CASE outputState OF
	eSpecialStates.SLAVE_ENTER_PROCEDURE:
		bSerialTransition := clamper^.Execute(eCylinderCommands.COMMAND_B); //release
	16#201:
		//wait until trigger off
		bSerialTransition := NOT handy;
		IF bSerialTransition THEN
			SlotBase^.Valid := FALSE; //reset
		END_IF
		//
		IF toggleClear AND materialRemains = 0 THEN
			toggleClear := FALSE;
		END_IF
	16#202:
		//conditions
		//1. bypassed
		//2. handy on
		//3. toggle clear
		//4. material existed with light screen off
		IF toggleClear OR bIsBypassed OR handy OR ( lightScreen AND SlotBase^.Valid) THEN
			bSerialTransition := TRUE;
		END_IF
		//once material detected , clamper imdiatly
		IF NOT SlotBase^.Valid AND materialValidSensor THEN
			clamper^.Execute(eCylinderCommands.COMMAND_A);
			SlotBase^.Valid := TRUE;
			//count-up
			inputCounter := inputCounter + 1;
			// material transfer
			SlotBase^.Act := TRUE;
		END_IF
	16#203:
		IF clamper^.Execute(eCylinderCommands.COMMAND_A) THEN
			//closure
			NextState := eSpecialStates.SLAVE_WORK_DONE;
		END_IF
END_CASE

METHOD FB_init : BOOL
VAR_INPUT
	bInitRetains : BOOL; // if TRUE, the retain variables are initialized (warm start / cold start)
	bInCopyCode : BOOL;  // if TRUE, the instance afterwards gets moved into the copy code (online change)
	
	argParent : POINTER TO RunUnitGeneric;
	argSlotBase : POINTER TO RunMaterial;
	argSlotLast : POINTER TO RunMaterial;
	
	argWorkingSignal : POINTER TO BOOL;
	
	argClamper : POINTER TO RunCylinder;
END_VAR
//initialize 
Parent := argParent;
SlotBase := argSlotBase;
SlotLast := argSlotLast;
//
IF bInitRetains THEN
	NextState := eSpecialStates.INITIAL_BEGIN;
END_IF

controller := Parent;

workingSignal := argWorkingSignal; //link
//link
clamper := argClamper;
END_METHOD

METHOD Initialize : BOOL
VAR_INPUT
END_VAR

CASE outputState OF
	eSpecialStates.INITIAL_BEGIN:
		IF clamper^.Execute(eCylinderCommands.COMMAND_A) THEN
			//release clamper
			NextState := eSpecialStates.INITIAL_END;
		END_IF
END_CASE

Initialize := SUPER^.Initialize();
END_METHOD

END_FUNCTION_BLOCK

// ---- POUs/Stations/RunUnitCellularAIO.TcPOU
FUNCTION_BLOCK RunUnitCellularAIO EXTENDS RunUnitIndexerMaster
VAR_INPUT
	allHit : BOOL;
	allReach : BOOL;
	allRelease : BOOL;
END_VAR
VAR_OUTPUT
	triggerHit : BOOL;
	triggerRelease : BOOL;
END_VAR
VAR
	ioConveyor : POINTER TO ioBundleConveyor;
	runTimer : TON;
END_VAR
VAR PERSISTENT
	//Checkpoints
	commandTriggerRaise: TIME; //trigger point
	commandReceivingTime : TIME; //if not all lifter done until then , slowdown conveyor motion
END_VAR

//implement state 3
isLastSlotOccupied := TRUE; //always pass carreir even empty material

SUPER^(); //run indexer master

IF bSerialTransition AND State = 1 THEN
	NextState := 16#10; //state override : release lifters
END_IF
IF bSerialTransition AND state=2 THEN
	//moving
	//timer setup and run
	runTimer.IN := TRUE;
	runTimer.PT := commandTriggerRaise;
	ioConveyor^.run := TRUE;

	NextState := 16#11; //re-direct
END_IF

CASE outputState OF
	//-------------------------release lifters
	16#10:
	IF allRelease THEN
		//reset
		triggerRelease:=FALSE;				
		NextState := 2; //wait syncAckowledged 
	END_IF
	//------------------start running
	16#11:
	IF runTimer.Q THEN	
		triggerHit := TRUE;//until trigger raise reached , trigger all lifter to move
		bSerialTransition:= TRUE; //serial transition
		
		runTimer.IN := FALSE;
	ELSE
		//on-going , not trigger lifter
	END_IF
	16#12:
	IF allHit THEN
		triggerHit:=FALSE;
		syncEngaged := FALSE ;// sending over
		bSerialTransition:= TRUE; //serial transition
	ELSIF timeoutTimer.Q THEN
		//sending error , raising alarm
		AlarmCode := eErrorCodes.AC_CONVEYOR_JAMMED;
	END_IF
	16#13:
	IF allReach THEN	
		bSerialTransition := TRUE; //since working signal raised by individual lifter?
	ELSIF timeoutTimer.Q THEN	
		//receiving error , should stop conveyor	
		AlarmCode := eErrorCodes.AC_CONVEYOR_NOT_REACHED;
	END_IF
	16#14:
	IF Upstream<>0 AND_THEN Upstream^.syncEngaged THEN
		//receive data
		SlotBase^.Valid := Upstream^.syncMatValid;
		SlotBase^.Id := Upstream^.syncMatId;
		//After all reached , then pull upstream
		Upstream^.syncAcknowledged := TRUE;//pull upstream when ready
		bSerialTransition:= TRUE; //serial transition	
	ELSIF timeoutTimer.Q THEN 
		//waiting upstream , reminder
	END_IF
	16#15:
	//wait until upstream action done
	bSerialTransition := Upstream<>0 AND_THEN NOT Upstream^.syncEngaged;
	IF bSerialTransition THEN
		//start count-down
		runTimer.PT := commandReceivingTime;
		runTimer.IN := TRUE;
	ELSIF NOT bSerialTransition AND timeoutTimer.Q THEN
		//reminder	
	END_IF
	16#16:
	// on extension , only one oppertunity
	IF runTimer.Q THEN
		runTimer.IN := FALSE;
		ioConveyor^.run := FALSE; //conveyor stopped
		
		triggerRelease:=TRUE;
		Upstream^.syncAcknowledged := FALSE; //inform done
		
		NextState := 0;//done
	ELSE
		//wait motion done	
	END_IF	
	//------------------------end of running
END_CASE
//run timer
runTimer(IN:= , PT:= , Q=> , ET=> );

METHOD ConfigureRead : CellDataBlock
VAR_INPUT
	input : CellDataBlock;
	mode : eModes;
END_VAR
CASE input.unit.config.configId OF 
	0:
		ConfigureRead.unit.config.value := TO_DWORD(commandTriggerRaise);
	1:
		 ConfigureRead.unit.config.value:= TO_DWORD(commandReceivingTime);
	
END_CASE
END_METHOD

METHOD ConfigureWrite : BOOL
VAR_INPUT
	input : CellDataBlock;
	mode : eModes;
END_VAR
CASE input.unit.config.configId OF 
	0:
		commandTriggerRaise := TO_TIME(input.unit.config.value);
	1:
		commandReceivingTime := TO_TIME(input.unit.config.value);
	
END_CASE
END_METHOD

METHOD FB_init : BOOL
VAR_INPUT
	bInitRetains : BOOL; // if TRUE, the retain variables are initialized (warm start / cold start)
	bInCopyCode : BOOL;  // if TRUE, the instance afterwards gets moved into the copy code (online change)
	
	argParent : POINTER TO RunUnitGeneric;
	argSlotBase : POINTER TO RunMaterial;
	argSlotLast : POINTER TO RunMaterial;
	
	argUpstream : POINTER TO RunUnitTransporterBase;
	argAxis : POINTER TO RunAxis;

	argIo : pointer to ioBundleConveyor;
END_VAR
//initialize 
Parent := argParent;
SlotBase := argSlotBase;
SlotLast := argSlotLast;

Axis := 0; //no servo axis
Upstream := argUpstream;

ioConveyor := argIo;
END_METHOD

METHOD Initialize : BOOL
VAR_INPUT
END_VAR
//direct change state
NextState := eSpecialStates.INITIAL_END;
Initialize := SUPER^.Initialize();
END_METHOD

END_FUNCTION_BLOCK

// ---- POUs/Stations/RunUnitCellularC.TcPOU
FUNCTION_BLOCK RunUnitCellularC EXTENDS RunUnitTransporterBase
VAR_INPUT
END_VAR
VAR_OUTPUT
END_VAR
VAR
	//devices
	reachSensor : POINTER TO RunSignal;
	interfereSensor : POINTER TO RunSignal;
	holderCylinder : POINTER TO RunCylinder;
	pusherCylinder : POINTER TO RunCylinder;
	//liner
	liner : POINTER TO RunAxis;
	ptLinerSend : POINTER TO ParameterSet;
	ptLinerWork : POINTER TO ParameterSet;
	ptLinerReceive : POINTER TO ParameterSet;
	//rotator (option
	rotator : POINTER TO RunAxis;
	ptRotatorMutual : POINTER TO ParameterSet;
	ptRotatorSend : POINTER TO ParameterSet;
	ptRotatorReceive : POINTER TO ParameterSet;
END_VAR
VAR PERSISTENT
	//TODO memorize carrier existed?
	isQuery : bool ; //whether query material data when material income
END_VAR

SUPER^();
//inherits sync/mat relative variables

//interfere auto cut axis	(high priority


CASE outputState OF 
	eSpecialStates.INITIAL_BEGIN:
		bSerialTransition := holderCylinder^.Execute(eCylinderCommands.COMMAND_B); //hold
	eSpecialStates.INITIAL_STATE_1:
		IF (rotator=0 OR (rotator<>0 AND_THEN rotator^.ExecuteParameter(ptRotatorMutual))) THEN
			NextState := eSpecialStates.INITIAL_END;
		END_IF
	//-----------------switch function
	0:
		IF reachSensor^.debouncedOn THEN
			//occupied , sending procedure
			NextState := 16#2000;
		ELSE
			//vacuumed , receiving procedure
			NextState := 16#1000;
		END_IF
	//-----------------sending procedure 
	16#2000:
		IF holderCylinder^.Execute(eCylinderCommands.COMMAND_B) AND NOT transitionByte.0 THEN
			transitionByte.0 := TRUE;
		END_IF
		IF pusherCylinder^.Execute(eCylinderCommands.COMMAND_A) AND NOT transitionByte.1 THEN
			transitionByte.1 := TRUE;
		END_IF
		IF transitionByte = 16#3 AND interfereSensor^.debouncedOff THEN
			bSerialTransition := TRUE;
		END_IF
	16#2001:
		bSerialTransition := rotator=0 OR (rotator<>0 AND_THEN rotator^.ExecuteParameter(ptRotatorMutual)); //otherwise would interfere
	16#2002:
		bSerialTransition := liner^.ExecuteParameter(ptLinerSend);
	16#2003:
		bSerialTransition := rotator=0 OR (rotator<>0 AND_THEN rotator^.ExecuteParameter(ptRotatorSend)); //reached then rotate
	16#2004:
		IF holderCylinder^.Execute(eCylinderCommands.COMMAND_A) THEN
			//release , wait to send
			IF SlotBase<>0 THEN
				syncMatValid := SlotBase^.Valid;
				syncMatId := SlotBase^.Id;
			END_IF			
			syncEngaged := TRUE;
			bSerialTransition := TRUE;
		END_IF
	16#2005:
		IF syncAcknowledged AND_THEN pusherCylinder^.Execute(eCylinderCommands.COMMAND_B) THEN
			//go out
			bSerialTransition := TRUE;
		END_IF
	16#2006:
		IF interfereSensor^.debouncedOff AND reachSensor^.debouncedOff THEN
			syncEngaged := FALSE;//leaved
			bSerialTransition := TRUE;
		END_IF
	16#2007:
		IF pusherCylinder^.Execute(eCylinderCommands.COMMAND_A) AND NOT syncAcknowledged THEN
			//make sure synchronized
			NextState := 16#1000; //rewind
		END_IF
	//---------------------receiving procedure
	16#1000:
		// holder off , pusher off , rotator/linear in receive position
		IF NOT transitionByte.0 AND_THEN holderCylinder^.Execute(eCylinderCommands.COMMAND_A) THEN
			transitionByte.0 := TRUE;
		END_IF
		IF  NOT transitionByte.1  AND_THEN pusherCylinder^.Execute(eCylinderCommands.COMMAND_A) THEN
			transitionByte.1 := TRUE;
		END_IF
		IF NOT transitionByte.2 AND_THEN (rotator=0 OR (rotator<>0 AND_THEN rotator^.ExecuteParameter(ptRotatorMutual))) THEN
			transitionByte.2 := TRUE;
		END_IF		
		IF transitionByte = 16#7 AND interfereSensor^.debouncedOff THEN
			bSerialTransition := TRUE;
		END_IF
	16#1001:
		bSerialTransition := liner^.ExecuteParameter(ptLinerReceive);
	16#1002:
			bSerialTransition := rotator=0 OR (rotator<>0 AND_THEN rotator^.ExecuteParameter(ptRotatorReceive));
	16#1003:
		IF Upstream<>0 AND_THEN Upstream^.syncEngaged THEN
			//receive data
			IF SlotBase<>0 THEN
				SlotBase^.Valid := Upstream^.syncMatValid;
				SlotBase^.Id := Upstream^.syncMatId;
			END_IF		
			//reply
			Upstream^.syncAcknowledged := TRUE; //
			bSerialTransition := TRUE;
		END_IF
	16#1004:
		bSerialTransition := interfereSensor^.debouncedOff AND reachSensor^.debouncedOn;
		IF  bSerialTransition THEN
			SlotBase^.Act := isQuery;
		END_IF
	16#1005:
		IF Upstream<>0 AND_THEN NOT Upstream^.syncEngaged THEN
			Upstream^.syncAcknowledged := FALSE; //completely follow upstream ,
			bSerialTransition := TRUE;
		END_IF
	16#1006:
		IF holderCylinder^.Execute(eCylinderCommands.COMMAND_B) THEN
			NextState := 16#3000;
		END_IF
	//------------------Work
	16#3000:
		IF NOT bSerialTransition AND_THEN (rotator=0 OR (rotator<>0 AND_THEN rotator^.ExecuteParameter(ptRotatorMutual))) THEN
			bSerialTransition := TRUE;
		END_IF
	16#3001:	
		IF NOT transitionByte.0 AND_THEN liner^.ExecuteParameter(ptLinerWork) THEN
			transitionByte.0 := TRUE;	
		END_IF
		transitionByte.1 := NOT SlotBase^.Act;
		IF transitionByte = 3 THEN
			slaveWorkingSignal[1] := slaveLinkageStatus[1]; //start working
			bSerialTransition := TRUE;
		END_IF
	16#3002:
		IF NOT slaveWorkingSignal[1] THEN
			NextState := 16#2000;
		END_IF
END_CASE

METHOD FB_init : BOOL
VAR_INPUT
	bInitRetains : BOOL; // if TRUE, the retain variables are initialized (warm start / cold start)
	bInCopyCode : BOOL;  // if TRUE, the instance afterwards gets moved into the copy code (online change)
	
	argParent : POINTER TO RunUnitGeneric;
	argSlotBase : POINTER TO RunMaterial;
	argSlotLast : POINTER TO RunMaterial;
	
	argUpstream : POINTER TO RunUnitTransporterBase;
	
	argLinear : POINTER TO RunAxis;
	argRotator : POINTER TO RunAxis;
	argReachSensor : POINTER TO RunSignal;
	argInterfereSensor : POINTER TO RunSignal;
	argHolderCylinder : POINTER TO RunCylinder;
	argPusherCylinder : POINTER TO RunCylinder;
END_VAR
VAR CONSTANT
	indexSend : INT := 1;
	indexReceive : INT := 2;
	indexMutual : INT := 3; //equals to work position to Cellular D
END_VAR
//initialize 
Parent := argParent;
SlotBase := argSlotBase;
SlotLast := argSlotLast;

Upstream := argUpstream;

IF Upstream=0 THEN
	isProxyMode:=TRUE; //no upstream , i am proxy
END_IF

//device link
liner := argLinear;

reachSensor := argReachSensor;
interfereSensor := argInterfereSensor;
holderCylinder := argHolderCylinder;
pusherCylinder := argPusherCylinder;
//position link
ptLinerSend := ADR(liner^.ptpCommands[indexSend]);
ptLinerReceive := ADR(liner^.ptpCommands[indexReceive]);
ptLinerWork := ADR(liner^.ptpCommands[indexMutual]);
// rotator(option
IF argRotator <> 0 THEN
	rotator := argRotator;
	
	ptRotatorSend := ADR(rotator^.ptpCommands[indexSend]);
	ptRotatorReceive := ADR(rotator^.ptpCommands[indexReceive]);
	ptRotatorMutual := ADR(rotator^.ptpCommands[indexMutual]);
END_IF
END_METHOD

END_FUNCTION_BLOCK

// ---- POUs/Stations/RunLifterCelluar.TcPOU
FUNCTION_BLOCK RunLifterCelluar EXTENDS RunUnitGeneric
VAR_INPUT
	//sensor
	ptObstacleSensorStatus : POINTER TO BOOL; //fibers
	ptReachSensorStatus : POINTER TO BOOL; //approximities
END_VAR
VAR_OUTPUT
END_VAR
VAR	
	mHit : BOOL ;
	mRelease : BOOL;	

	//actuator
	//axis
	AxisVertical : POINTER TO RunAxis;
	AxisHorizon : POINTER TO RunAxis;
	//cylinder
	Cylinder : POINTER TO RunCylinder;
	
	//carrier mover(vertical
	ptCommandLifterHit : POINTER TO ParameterSet; // raise to hit
	ptCommandLifterRelease : POINTER TO ParameterSet; //release
	ptCommandLifterWorking : POINTER TO ParameterSet; //lift carrier to working position
	//carrier mover(horizon
	ptCommandHorizonHit : POINTER TO ParameterSet;
	ptCommandHorizonWorking : POINTER TO ParameterSet;
	
	
	isAllWorkDone : BOOL; //dispatch work to working station
	nCounter : int ;
END_VAR

SUPER^();

CASE outputState OF
	//-------------------------Initialize
	eSpecialStates.INITIAL_BEGIN:
		bSerialTransition:=Cylinder^.Execute(eCylinderCommands.COMMAND_A);//MC on would be taken by method call
	eSpecialStates.INITIAL_STATE_1:
		bSerialTransition :=  AxisVertical^.ExecuteParameter(ptCommandLifterRelease);
	eSpecialStates.INITIAL_STATE_2:
		IF AxisHorizon=0 OR (AxisHorizon<>0 AND_THEN AxisHorizon^.ExecuteParameter(ptCommandHorizonHit)) THEN
			NextState := eSpecialStates.INITIAL_END;
		END_IF
	//-------------------------Hit
	0:
	//initiale state : 
	// 1. axis in release position
	// 2. cylinder  in A
	// 3. all sensor off
	bSerialTransition := mHit AND NOT ptObstacleSensorStatus^ ;//if execute flag on
	atomicOperation := bSerialTransition; //once satisfied , do not be interrupted (on-the-fly operation
	1:
	bSerialTransition := AxisVertical^.ExecuteParameter(ptBlock:=ptCommandLifterHit);
	IF bSerialTransition THEN
		mHit := FALSE; //reset
		atomicOperation := FALSE; //release
	END_IF
	2:
	//once reach sensor detected , n
	bSerialTransition := ptReachSensorStatus^;	
	3:
	//to working position
	bSerialTransition := AxisVertical^.ExecuteParameter(ptCommandLifterWorking);
	4:
	//hold
	bSerialTransition := Cylinder^.Execute(eCylinderCommands.COMMAND_B);
	5:
	//to working position
	IF AxisHorizon=0 OR (AxisHorizon<>0 AND_THEN AxisHorizon^.ExecuteParameter(ptCommandHorizonWorking)) THEN
		//dispatching work to station
		//Dispatch working signal to all station
		FOR nCounter := 1 TO 4 BY 1 DO
		  slaveWorkingSignal[nCounter]	:= slaveLinkageStatus[nCounter];
		END_FOR
		NextState := 16#10;
	END_IF
	//---------------------------releasing
	16#20:
	bSerialTransition := mRelease;
	IF bSerialTransition THEN
		mRelease := FALSE;
	END_IF
	16#21:
	bSerialTransition := AxisHorizon=0 OR (AxisHorizon<>0 AND_THEN  AxisHorizon^.ExecuteParameter(ptCommandHorizonHit));
	16#22:	
	bSerialTransition := Cylinder^.Execute(eCylinderCommands.COMMAND_A);	//release holder
	16#23:
	bSerialTransition :=  AxisVertical^.ExecuteParameter(ptCommandLifterRelease);
	16#24:
	IF NOT ptReachSensorStatus^ THEN
		//make sure all state reseted
		NextState := 0;
	END_IF
	
	//----------------------------- working
	16#10:
		//check if all working signal off
		isAllWorkDone := TRUE;
		FOR nCounter :=1 TO 4 BY 1 DO
			isAllWorkDone := isAllWorkDone AND  not slaveWorkingSignal[nCounter];
		END_FOR
		IF isAllWorkDone THEN
			NextState := 16#20;
		END_IF
END_CASE

METHOD FB_init : BOOL
VAR_INPUT
	bInitRetains : BOOL; // if TRUE, the retain variables are initialized (warm start / cold start)
	bInCopyCode : BOOL;  // if TRUE, the instance afterwards gets moved into the copy code (online change)

	argParent : POINTER TO RunUnitGeneric;
	argSlotBase : POINTER TO RunMaterial;
	argSlotLast : POINTER TO RunMaterial;
	
	argAxisVertical : POINTER TO RunAxis;
	argAxisHorizon : POINTER TO RunAxis;
	argCylinder : POINTER TO RunCylinder;
	
	argObstacleSensor : POINTER TO RunSignal;
	argReachSensor : POINTER TO RunSignal;
	
END_VAR
VAR CONSTANT
	indexRelease : INT := 3;
	indexHit : INT := 1;
	indexWorking : INT := 2;
END_VAR
//initialize 
Parent := argParent;
SlotBase := argSlotBase;
SlotLast := argSlotLast;

//initializing , link related commandblock/sensor/cylinder


//actuator
	//axis
AxisVertical := argAxisVertical;
AxisHorizon := argAxisHorizon;
//cylinder
Cylinder := argCylinder;
	
//lifter
ptCommandLifterHit := ADR(AxisVertical^.ptpCommands[indexHit]); // raise to hit
ptCommandLifterRelease :=  ADR(AxisVertical^.ptpCommands[indexRelease]);; //release
ptCommandLifterWorking :=  ADR(AxisVertical^.ptpCommands[indexWorking]);; //lift carrier to working position
//horizon
ptCommandHorizonWorking := ADR(AxisHorizon^.ptpCommands[indexWorking]);
ptCommandHorizonHit :=ADR(AxisHorizon^.ptpCommands[indexHit]);
//sensor
ptObstacleSensorStatus := ADR(argObstacleSensor^.debouncedOn); //fibers
ptReachSensorStatus :=ADR(argReachSensor^.debouncedOn); //approximities
END_METHOD

PROPERTY IsHit : BOOL
GET
IsHit:=(State>=2);
END_GET
SET
mHit:=IsHit;
END_SET
END_PROPERTY

PROPERTY IsReach : BOOL
GET
IsReach:=(State >=3);
END_GET
SET
END_SET
END_PROPERTY

PROPERTY IsReleased : BOOL
GET
IsReleased:=(State=0);
END_GET
SET
mRelease := isReleased;
END_SET
END_PROPERTY

END_FUNCTION_BLOCK

// ---- POUs/Stations/RunUnitCellularA.TcPOU
FUNCTION_BLOCK RunUnitCellularA EXTENDS RunUnitIndexerMaster
VAR_INPUT
	allHit : BOOL;
	allReach : BOOL;
	allRelease : BOOL;
END_VAR
VAR_OUTPUT
	triggerHit : BOOL;
	triggerRelease : BOOL;
END_VAR
VAR
	// conveyor related 
	ptCommandFast : POINTER TO ParameterSet; // as error stop position (jammed
	ptCommandSlow : POINTER TO ParameterSet; // as Pitch1
	
	//Checkpoints
	commandTriggerRaise: ParameterSet; //trigger point
	commandCheckRaise : ParameterSet; //if not all lifter done until then , slowdown conveyor motion
	//Lifters
	//lifters : ARRAY[1..3] OF POINTER TO RunLifterCelluar;
	commandSetZero : ParameterSet;
	commandFinalGoal : ParameterSet;
	ptCommandPitch2 : POINTER TO ParameterSet;

	fastExecute : BOOL;
	slowExecute : BOOL;
	finalGoalExecute : BOOL;
	
	fastDone : BOOL;
	slowDone: BOOL;
	finalGoalDone : BOOL;
			
END_VAR

//implement state 3
isLastSlotOccupied := TRUE; //always pass carreir even empty material

SUPER^(); //run indexer master

//----------------------
//Conveyor buffer modes
//----------------------
IF NOT fastDone AND fastExecute THEN
	fastDone := Axis^.ExecuteParameterBuffer(ptCommandFast,
	bufferIndex:=1);
END_IF
IF NOT slowDone AND slowExecute THEN
	slowDone := Axis^.ExecuteParameterBuffer(ptCommandSlow,
	bufferIndex:=2);
END_IF
IF NOT finalGoalDone AND finalGoalExecute THEN
	finalGoalDone := Axis^.ExecuteParameterBuffer(ADR(commandFinalGoal),
	bufferIndex:=3);
END_IF

IF bSerialTransition AND State = 1 THEN
	NextState := 16#10; //state override : release lifters
END_IF
//-----------------------------
// On-the-fly trigger upstream
//-----------------------------
IF State >=3 AND State <=6 AND_THEN Upstream<>0 AND Upstream^.syncEngaged AND NOT Upstream^.syncAcknowledged THEN
	//receive data
	SlotBase^.Id := Upstream^.syncMatId;
	SlotBase^.Valid := Upstream^.syncMatValid;
	//reply	
	Upstream^.syncAcknowledged := TRUE;//pull upstream when ready
	//set-up final goal
	commandFinalGoal.command := eCommandTypes.POSITION;
	commandFinalGoal.parameter.position.Velocity := ptCommandPitch2^.parameter.position.Velocity;
	commandFinalGoal.parameter.position.Acceleration := ptCommandPitch2^.parameter.position.Acceleration;
	commandFinalGoal.parameter.position.Deceleration := ptCommandPitch2^.parameter.position.Deceleration;
	commandFinalGoal.parameter.position.Position := Axis^.PositionFeedback + ptCommandPitch2^.parameter.position.Position; //goal extended
	
	//prevent backward
	IF commandFinalGoal.parameter.position.Position < ptCommandSlow^.parameter.position.Position THEN
		commandFinalGoal.parameter.position.Position := ptCommandSlow^.parameter.position.Position;
	END_IF
	//entered atomic operation , do not interrupt
	atomicOperation:=TRUE;
END_IF
//once alarm occured , release atomic 
IF atomicOperation AND AlarmCode<>0 THEN
	atomicOperation := FALSE; 
END_IF

CASE outputState OF
	//-------------------------release lifters
	16#10:
	commandSetZero.command := eCommandTypes.SET_POSITION;
	commandSetZero.parameter.position.Position := 0;
	
	IF NOT transitionByte.0 THEN
		transitionByte.0 := Axis^.ExecuteParameter(ptBlock:= ADR(commandSetZero));//reset pos command to zero
	END_IF
	
	IF allRelease AND transitionByte.0 THEN
		//reset all 	
		fastExecute := FALSE;
		slowExecute := FALSE;
		finalGoalExecute:=FALSE;

		fastDone := FALSE;
		slowDone := FALSE;
		finalGoalDone:=FALSE;	
	
		triggerRelease:=FALSE;
		
		//before enter deceleration
		commandCheckRaise.parameter.position.Position := (ptCommandFast^.parameter.position.Velocity * ptCommandFast^.parameter.position.Velocity);
		commandCheckRaise.parameter.position.Position := commandCheckRaise.parameter.position.Position / (ptCommandFast^.parameter.position.Deceleration * 1.8);
		
		NextState:=2; //merge back default sequence
	END_IF
	//------------------start running
	3:
	fastExecute := TRUE; //start to go
	bSerialTransition:= TRUE; //serial transition
	4:
	IF Axis^.PositionFeedback >= commandTriggerRaise.parameter.position.Position THEN		
		triggerHit := TRUE;//until trigger raise reached , trigger all lifter to move
		bSerialTransition:= TRUE; //serial transition
	//Else : on-going , not trigger lifter
	END_IF
	5:
	IF Axis^.PositionFeedback >= commandCheckRaise.parameter.position.Position THEN
		IF allHit THEN
			triggerHit:=false;
			slowExecute:=TRUE;//able to slowdown to bump
			syncEngaged := false ;// sending over
			bSerialTransition:= TRUE; //serial transition
		ELSIF fastDone THEN
			//fast had executed , but not all hit , trigger alarm (stop doing next move
			AlarmCode := eErrorCodes.AC_CONVEYOR_JAMMED;
		END_IF
	//Else : on going , not reached the check point
	END_IF
	6:
	IF Upstream<>0 AND_THEN Upstream^.syncAcknowledged AND fastDone THEN
		//wait first command block done , otherwise would raise 0x4292 (buffer fulled)
		finalGoalExecute:=TRUE;//need do extension
		bSerialTransition:= TRUE; //serial transition	
	ELSIF allReach THEN
		//manually put carrier in?
	END_IF
	//---------------------------------------------
	7:
	// on extension , only one oppertunity
	bSerialTransition := finalGoalDone;
	//------------------------end of running
	8:
	IF allReach THEN
		triggerRelease:=TRUE; //for those already done , able to release
		bSerialTransition := TRUE;
	ELSE
		AlarmCode := eErrorCodes.AC_CONVEYOR_NOT_REACHED;
	END_IF
	9:
	IF Upstream <> 0 AND_THEN NOT Upstream^.syncEngaged THEN
		Upstream^.syncAcknowledged := FALSE; // received carrier
		NextState :=0; //back to check if all MatSync done
	ELSE
		// upstream not synchroized			
	END_IF
END_CASE

METHOD FB_init : BOOL
VAR_INPUT
	bInitRetains : BOOL; // if TRUE, the retain variables are initialized (warm start / cold start)
	bInCopyCode : BOOL;  // if TRUE, the instance afterwards gets moved into the copy code (online change)
	
	argParent : POINTER TO RunUnitGeneric;
	argSlotBase : POINTER TO RunMaterial;
	argSlotLast : POINTER TO RunMaterial;
	
	argUpstream : POINTER TO RunUnitTransporterBase;
	argAxis : POINTER TO RunAxis;

END_VAR
VAR CONSTANT
	indexFast : INT := 1;
	indexSlow : INT := 2;
	indexComp : INT := 3;
END_VAR
//initialize 
Parent := argParent;
SlotBase := argSlotBase;
SlotLast := argSlotLast;

Axis := argAxis;
Upstream := argUpstream;

//
IF Axis<>0 THEN
	ptCommandFast := ADR(Axis^.ptpCommands[indexFast]);
	ptCommandSlow := ADR(Axis^.ptpCommands[indexSlow]);
	ptCommandPitch2 := ADR(Axis^.ptpCommands[indexComp]);
	commandTriggerRaise.parameter.position.Position := 250; //carrier length
END_IF

IF Upstream=0 THEN
	isProxyMode:=TRUE; //no upstream , i am proxy
END_IF
END_METHOD

END_FUNCTION_BLOCK

// ---- POUs/Stations/RunUnitDummy.TcPOU
FUNCTION_BLOCK RunUnitDummy EXTENDS RunUnitSlave
VAR_INPUT
END_VAR
VAR_OUTPUT
END_VAR
VAR
END_VAR
VAR PERSISTENT
	var1 : INT := 1;
	var2 : INT := 2;
END_VAR

SUPER^();

METHOD ConfigureRead : CellDataBlock
VAR_INPUT
	input : CellDataBlock;
	mode : eModes;
END_VAR
//ConfigureRead := input;
CASE input.unit.config.configId OF
	0:
		 ConfigureRead.unit.config.value := TO_WORD(var1);
	1:
		ConfigureRead.unit.config.value := TO_WORD(var2);
END_CASE
END_METHOD

METHOD ConfigureWrite : BOOL
VAR_INPUT
	input : CellDataBlock;
	mode : eModes;
END_VAR
CASE input.unit.config.configId OF
	0:
		var1 := TO_INT(input.unit.config.value);
	1:
		var2 := TO_INT(input.unit.config.value);
END_CASE
END_METHOD

METHOD Initialize : BOOL
VAR_INPUT
END_VAR
CASE outputState OF
	eSpecialStates.INITIAL_BEGIN:		
			NextState := eSpecialStates.INITIAL_END;
END_CASE

Initialize := SUPER^.Initialize();
END_METHOD

END_FUNCTION_BLOCK
